TYPE ST_FB_MGMT_Steuerung :
STRUCT
	Freigabe			         : ST_Steuerung_auto_manu_BOOL;
	Freigabe_Deakt		: ST_Steuerung_auto_manu_BOOL;
	Betrieb_Anford		: ST_Steuerung_auto_manu_opti_BOOL;

	Regelung_Modus		: ST_Steuerung_auto_manu_opti_SINT;
	Regelung_Sollw		: ST_Steuerung_auto_manu_opti_REAL;
	Regelung_Sollw_Max	: ST_Steuerung_auto_manu_opti_REAL;
	Regelung_Sollw_Min	: ST_Steuerung_auto_manu_opti_REAL;

	Quittierung			: BOOL;

END_STRUCT
END_TYPE

(* stored: Version 1.1.0.1, ProductVersion 3.1.4024.9
   DUT ST_FB_MGMT_Steuerung: Id {e21e8640-b605-43fb-861a-fd571a350675} *)
